// TIA Portal V17 export
// export: Created 2025-03-10T13:12:20.1816657Z, ExportSetting WithDefaults, DisplayName Totally Integrated Automation Portal, DisplayVersion V17 Update 8, DisplayName TIA Portal Openness, DisplayVersion V17 Update 8, DisplayName TIA Portal Version Control Interface, DisplayVersion V17, DisplayName SINAMICS Startdrive Advanced, DisplayVersion V17 SP2, DisplayName SINAMICS Startdrive G110M, G120, G120C, G120D, G120P, G115D, DisplayVersion V17 SP2, DisplayName SINAMICS Startdrive G130, G150, S120, S150, SINAMICS MV, S210, DisplayVersion V17 SP2, DisplayName STEP 7 Professional, DisplayVersion V17 Update 8, DisplayName SINUMERIK ONE STEP 7 Toolbox, DisplayVersion V17 Update 12, DisplayName SINUMERIK 840D sl STEP 7 Toolbox, DisplayVersion V17 Update 12, DisplayName STEP 7 Safety, DisplayVersion V17 Update 6, DisplayName WinCC Advanced, DisplayVersion V17 Update 8
TYPE "COOLING_SENSOR"
// stored: IsFailsafeCompliant false
   STRUCT
      COOLING_FLOW_SENSOR_ACTUAL_VALUE : Real;   // COOLING FLOW SENSOR VALUE
      COOLING_TEMP_SENSOR_ACTUAL_VALUE : Real;   // COOLING TEMPERATURE SENSOR VALUE
      COOLING_FLOW_LOW_WARNING_HMI_VALUE : Real := 3.2;   // COOLING FLOW LOW WARNING VALUE
      COOLING_FLOW_HIGH_WARNING_HMI_VALUE : Real := 4.8;   // COOLING FLOW HIGH WARNING VALUE
      COOLING_FLOW_LOW_ALARM_HMI_VALUE : Real := 3.2;   // COOLING FLOW LOW ALARM VALUE
      COOLING_FLOW_HIGH_ALARM_HMI_VALUE : Real := 6.0;   // COOLING FLOW HIGH ALARM VALUE
      COOLING_TEMP_LOW_WARNING_HMI_VALUE : Real := 27.0;   // COOLING TEMPERATURE LOW WARNING VALUE
      COOLING_TEMP_HIGH_WARNING_HMI_VALUE : Real := 40.0;   // COOLING TEMPERATURE HIGH WARNING VALUE
      COOLING_TEMP_LOW_ALARM_HMI_VALUE : Real := 27.0;   // COOLING TEMPERATURE LOW ALARM VALUE
      COOLING_TEMP_HIGH_ALARM_HMI_VALUE : Real := 40.0;   // COOLING TEMPERATURE HIGH ALARM VALUE
   END_STRUCT;
END_TYPE
